// TIA Portal V21 export
VAR_GLOBAL   // PLC tag table "OutputAnalogici"
END_VAR
